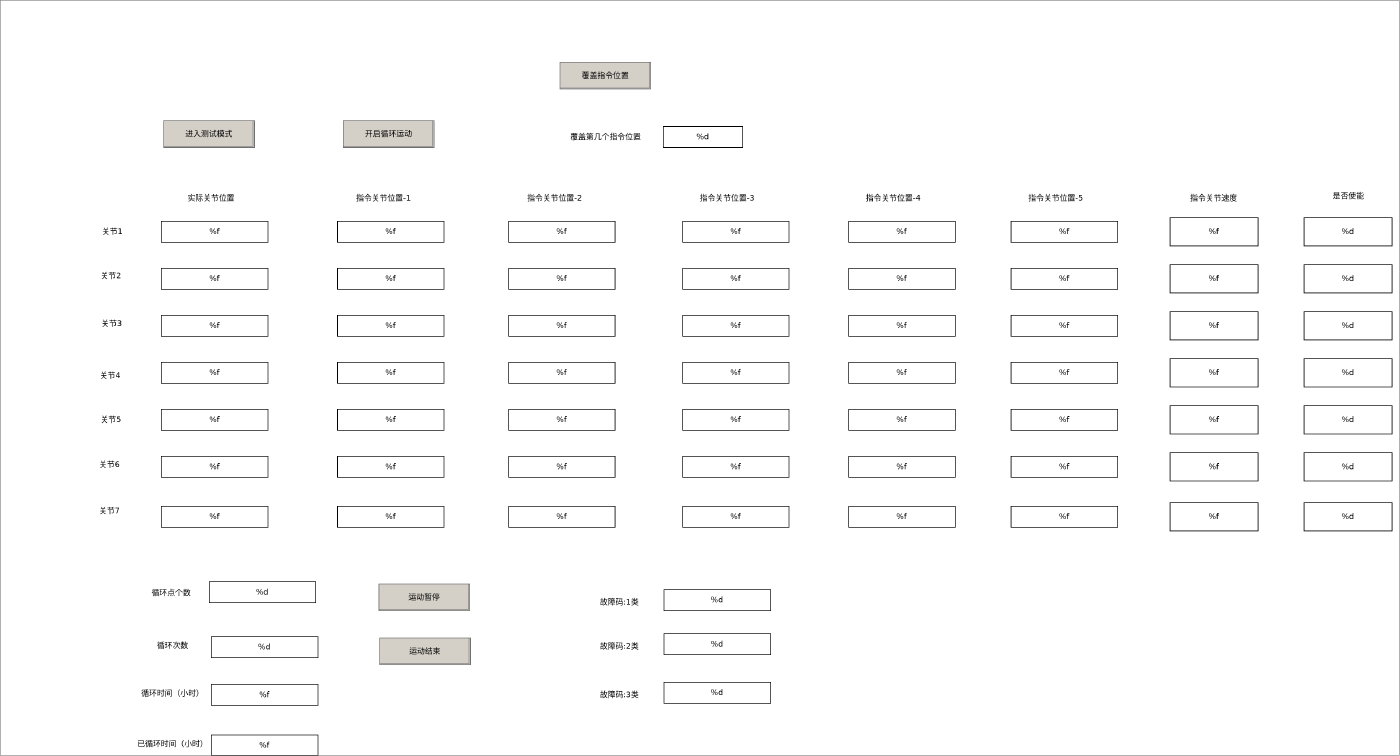
VISUALIZATION cycle_a1  // 1964x1061
    Label (221,263 150x30), "实际关节位置"
    Rectangle (226,310 150x30), "%f", text variable: g_cycleTest.m_armDHJntPos[1][1]
    Label (463,263 150x30), "指令关节位置-1"
    Button (229,169 128x38), "进入测试模式", colour toggle: g_cycleTest.m_enterCycleTestMode[1]
        toggle g_cycleTest.m_enterCycleTestMode[1]
    Button (481,169 128x38), "开启循环运动", colour toggle: g_cycleTest.m_startMotion[1]
        toggle g_cycleTest.m_startMotion[1]
    Rectangle (226,376 150x30), "%f", text variable: g_cycleTest.m_armDHJntPos[1][2]
    Rectangle (226,442 150x30), "%f", text variable: g_cycleTest.m_armDHJntPos[1][3]
    Rectangle (226,508 150x30), "%f", text variable: g_cycleTest.m_armDHJntPos[1][4]
    Rectangle (226,574 150x30), "%f", text variable: g_cycleTest.m_armDHJntPos[1][5]
    Rectangle (226,640 150x30), "%f", text variable: g_cycleTest.m_armDHJntPos[1][6]
    Rectangle (226,710 150x30), "%f", text variable: g_cycleTest.m_armDHJntPos[1][7]
    Rectangle (473,310 150x30), "%f", text variable: g_cycleTest.m_targetJntPos[1,1][1]
        OnMouseClick: write the text variable via Default
    Rectangle (473,376 150x30), "%f", text variable: g_cycleTest.m_targetJntPos[1,1][2]
        OnMouseClick: write the text variable via Default
    Rectangle (473,442 150x30), "%f", text variable: g_cycleTest.m_targetJntPos[1,1][3]
        OnMouseClick: write the text variable via Default
    Rectangle (473,508 150x30), "%f", text variable: g_cycleTest.m_targetJntPos[1,1][4]
        OnMouseClick: write the text variable via Default
    Rectangle (473,574 150x30), "%f", text variable: g_cycleTest.m_targetJntPos[1,1][5]
        OnMouseClick: write the text variable via Default
    Rectangle (473,640 150x30), "%f", text variable: g_cycleTest.m_targetJntPos[1,1][6]
        OnMouseClick: write the text variable via Default
    Rectangle (473,710 150x30), "%f", text variable: g_cycleTest.m_targetJntPos[1,1][7]
        OnMouseClick: write the text variable via Default
    Label (703,263 150x30), "指令关节位置-2"
    Rectangle (713,310 150x30), "%f", text variable: g_cycleTest.m_targetJntPos[1,2][1]
        OnMouseClick: write the text variable via Default
    Rectangle (713,376 150x30), "%f", text variable: g_cycleTest.m_targetJntPos[1,2][2]
        OnMouseClick: write the text variable via Default
    Rectangle (713,442 150x30), "%f", text variable: g_cycleTest.m_targetJntPos[1,2][3]
        OnMouseClick: write the text variable via Default
    Rectangle (713,508 150x30), "%f", text variable: g_cycleTest.m_targetJntPos[1,2][4]
        OnMouseClick: write the text variable via Default
    Rectangle (713,574 150x30), "%f", text variable: g_cycleTest.m_targetJntPos[1,2][5]
        OnMouseClick: write the text variable via Default
    Rectangle (713,640 150x30), "%f", text variable: g_cycleTest.m_targetJntPos[1,2][6]
        OnMouseClick: write the text variable via Default
    Rectangle (713,710 150x30), "%f", text variable: g_cycleTest.m_targetJntPos[1,2][7]
        OnMouseClick: write the text variable via Default
    Label (945,263 150x30), "指令关节位置-3"
    Rectangle (957,310 150x30), "%f", text variable: g_cycleTest.m_targetJntPos[1,3][1]
        OnMouseClick: write the text variable via Default
    Rectangle (957,376 150x30), "%f", text variable: g_cycleTest.m_targetJntPos[1,3][2]
        OnMouseClick: write the text variable via Default
    Rectangle (957,442 150x30), "%f", text variable: g_cycleTest.m_targetJntPos[1,3][3]
        OnMouseClick: write the text variable via Default
    Rectangle (957,508 150x30), "%f", text variable: g_cycleTest.m_targetJntPos[1,3][4]
        OnMouseClick: write the text variable via Default
    Rectangle (957,574 150x30), "%f", text variable: g_cycleTest.m_targetJntPos[1,3][5]
        OnMouseClick: write the text variable via Default
    Rectangle (957,640 150x30), "%f", text variable: g_cycleTest.m_targetJntPos[1,3][6]
        OnMouseClick: write the text variable via Default
    Rectangle (957,710 150x30), "%f", text variable: g_cycleTest.m_targetJntPos[1,3][7]
        OnMouseClick: write the text variable via Default
    Label (1178,263 150x30), "指令关节位置-4"
    Rectangle (1190,310 150x30), "%f", text variable: g_cycleTest.m_targetJntPos[1,4][1]
        OnMouseClick: write the text variable via Default
    Rectangle (1190,376 150x30), "%f", text variable: g_cycleTest.m_targetJntPos[1,4][2]
        OnMouseClick: write the text variable via Default
    Rectangle (1190,442 150x30), "%f", text variable: g_cycleTest.m_targetJntPos[1,4][3]
        OnMouseClick: write the text variable via Default
    Rectangle (1190,508 150x30), "%f", text variable: g_cycleTest.m_targetJntPos[1,4][4]
        OnMouseClick: write the text variable via Default
    Rectangle (1190,574 150x30), "%f", text variable: g_cycleTest.m_targetJntPos[1,4][5]
        OnMouseClick: write the text variable via Default
    Rectangle (1190,640 150x30), "%f", text variable: g_cycleTest.m_targetJntPos[1,4][6]
        OnMouseClick: write the text variable via Default
    Rectangle (1190,710 150x30), "%f", text variable: g_cycleTest.m_targetJntPos[1,4][7]
        OnMouseClick: write the text variable via Default
    Label (1406,263 150x30), "指令关节位置-5"
    Rectangle (1418,310 150x30), "%f", text variable: g_cycleTest.m_targetJntPos[1,5][1]
        OnMouseClick: write the text variable via Default
    Rectangle (1418,376 150x30), "%f", text variable: g_cycleTest.m_targetJntPos[1,5][2]
        OnMouseClick: write the text variable via Default
    Rectangle (1418,442 150x30), "%f", text variable: g_cycleTest.m_targetJntPos[1,5][3]
        OnMouseClick: write the text variable via Default
    Rectangle (1418,508 150x30), "%f", text variable: g_cycleTest.m_targetJntPos[1,5][4]
        OnMouseClick: write the text variable via Default
    Rectangle (1418,574 150x30), "%f", text variable: g_cycleTest.m_targetJntPos[1,5][5]
        OnMouseClick: write the text variable via Default
    Rectangle (1418,640 150x30), "%f", text variable: g_cycleTest.m_targetJntPos[1,5][6]
        OnMouseClick: write the text variable via Default
    Rectangle (1418,710 150x30), "%f", text variable: g_cycleTest.m_targetJntPos[1,5][7]
        OnMouseClick: write the text variable via Default
    Label (165,817 150x30), "循环点个数"
    Rectangle (293,816 150x30), "%d", text variable: g_cycleTest.m_pointSum[1]
        OnMouseClick: write the text variable via Default
    Rectangle (296,893 150x30), "%d", text variable: g_cycleTest.m_curCycleNum[1]
    Label (167,891 150x30), "循环次数"
    Button (531,819 128x38), "运动暂停", colour toggle: g_cycleTest.m_pause[1]
        toggle g_cycleTest.m_pause[1]
    Button (532,895 128x38), "运动结束", colour toggle: g_cycleTest.m_finish[1]
        toggle g_cycleTest.m_finish[1]
    Button (785,87 128x38), "覆盖指令位置", colour toggle: g_cycleTest.m_coverCmdPos[1]
        tap g_cycleTest.m_coverCmdPos[1]
    Rectangle (930,177 112x30), "%d", text variable: g_cycleTest.m_pntIdForCoverCmd[1]
        OnMouseClick: write the text variable via Default
    Label (777,178 145x28), "覆盖第几个指令位置"
    Label (1630,264 145x28), "指令关节速度"
    Rectangle (1641,305 124x40), "%f", text variable: g_cycleTest.m_targetJntVel[1][1]
        OnMouseClick: write the text variable via Default
    Rectangle (1641,371 124x40), "%f", text variable: g_cycleTest.m_targetJntVel[1][2]
        OnMouseClick: write the text variable via Default
    Rectangle (1641,437 124x40), "%f", text variable: g_cycleTest.m_targetJntVel[1][3]
        OnMouseClick: write the text variable via Default
    Rectangle (1641,503 124x40), "%f", text variable: g_cycleTest.m_targetJntVel[1][4]
        OnMouseClick: write the text variable via Default
    Rectangle (1641,569 124x40), "%f", text variable: g_cycleTest.m_targetJntVel[1][5]
        OnMouseClick: write the text variable via Default
    Rectangle (1641,635 124x40), "%f", text variable: g_cycleTest.m_targetJntVel[1][6]
        OnMouseClick: write the text variable via Default
    Rectangle (1641,705 124x40), "%f", text variable: g_cycleTest.m_targetJntVel[1][7]
        OnMouseClick: write the text variable via Default
    Rectangle (296,960 150x30), "%f", text variable: g_cycleTest.m_tgtCycleTime[1]
        OnMouseClick: write the text variable via Default
    Label (167,958 150x30), "循环时间（小时）"
    Rectangle (296,1031 150x30), "%f", text variable: g_cycleTest.m_curCycleTime[1]
        OnMouseClick: write the text variable via Default
    Label (167,1029 150x30), "已循环时间（小时）"
    Label (1819,261 145x28), "是否使能"
    Rectangle (1829,305 124x40), "%d", text variable: g_cycleTest.m_jntEnable[1][1]
        OnMouseClick: write the text variable via Default
    Rectangle (1829,371 124x40), "%d", text variable: g_cycleTest.m_jntEnable[1][2]
        OnMouseClick: write the text variable via Default
    Rectangle (1829,437 124x40), "%d", text variable: g_cycleTest.m_jntEnable[1][3]
        OnMouseClick: write the text variable via Default
    Rectangle (1829,503 124x40), "%d", text variable: g_cycleTest.m_jntEnable[1][4]
        OnMouseClick: write the text variable via Default
    Rectangle (1829,569 124x40), "%d", text variable: g_cycleTest.m_jntEnable[1][5]
        OnMouseClick: write the text variable via Default
    Rectangle (1829,635 124x40), "%d", text variable: g_cycleTest.m_jntEnable[1][6]
        OnMouseClick: write the text variable via Default
    Rectangle (1829,705 124x40), "%d", text variable: g_cycleTest.m_jntEnable[1][7]
        OnMouseClick: write the text variable via Default
    Label (106,307 103x36), "关节1"
    Label (104,369 103x36), "关节2"
    Label (105,436 103x36), "关节3"
    Label (103,509 103x36), "关节4"
    Label (104,571 103x36), "关节5"
    Label (102,634 103x36), "关节6"
    Label (102,699 103x36), "关节7"
    Rectangle (931,827 150x30), "%d", text variable: GVL_interactUI.g_errIdType1
        OnMouseClick: write the text variable via Default
    Label (794,830 150x30), "故障码:1类"
    Rectangle (931,889 150x30), "%d", text variable: GVL_interactUI.g_errIdType2
        OnMouseClick: write the text variable via Default
    Label (794,892 150x30), "故障码:2类"
    Rectangle (931,957 150x30), "%d", text variable: GVL_interactUI.g_errIdType3
        OnMouseClick: write the text variable via Default
    Label (794,960 150x30), "故障码:3类"
END_VISUALIZATION

(* stored: Version 1.1.0.1, ProductVersion 3.1.4024.11
   Visu cycle_a1: Id {f69d49d0-6778-47ae-aba0-4e1dfc9c085f} *)
